PROGRAM WritePersistentData
VAR

END_VAR

END_PROGRAM

(* stored: Version 1.1.0.1, ProductVersion 3.1.4024.10
   POU WritePersistentData: Id {2398b8ce-a0e3-4f23-861d-9cbd632541cb}, SpecialFunc None *)
